FUNCTION_BLOCK Fb_FeedingStateCheck
VAR_INPUT
	dut_FeedingState : FeedingState;
END_VAR
VAR_OUTPUT
	iReadableFeedingState : INT; // number which represent the state
END_VAR
VAR
	iBareNum : INT; // number we use to cycle through the FeedingState
	iLastFeedingState : FeedingState;
	
	nCaseNumberCycler : INT;
END_VAR

CASE nCaseNumberCycler OF
0: //Check if number is 0 or not. As 0 would represent initialized state
	//Also check whether it is there are any state changes or not
	IF (dut_FeedingState = iLastFeedingState ) THEN
		nCaseNumberCycler:=0;
	ELSE
		nCaseNumberCycler:=10;
	END_IF
	
10: //Cycling
	FOR iBareNum:=0 TO 11 BY 1 DO
		IF iBareNum < dut_FeedingState THEN
			iBareNum:=iBareNum+1;
		END_IF
		IF iBareNum > dut_FeedingState THEN
			iBareNum:=iBareNum-1;
		END_IF
		
	END_FOR
nCaseNumberCycler:=50;
50:	
nCaseNumberCycler:=0;
END_CASE

END_FUNCTION_BLOCK

(* stored: Version 1.1.0.1, ProductVersion 3.1.4024.12
   POU Fb_FeedingStateCheck: Id {8010df5e-b43a-4c51-8bc4-6969c2a277ea}, SpecialFunc None *)
